{attribute 'GeneratedUsingTerminal: EL6070-0000-0016'}
{attribute addProperty BoxType "EL6070-0000-0016"}
{attribute addProperty Id "InfoDataAT %I*InfoData_32EB74EA10"}
{attribute addProperty CRC "4004708084"}
{attribute addProperty Size "10"}
TYPE EL6070_EEB2FEF4 EXTENDS EtcSlaveTerminalBase_947E5A46 :
STRUCT
	{attribute addProperty Name "InfoData"}
	InfoData : InfoData_32EB74EA;
END_STRUCT
END_TYPE

(* stored: Version 1.2.0.0, ProductVersion 3.1.4024.9
   DUT EL6070_EEB2FEF4: Id {4efff1e7-fe69-4162-825a-c733cd3a4e45} *)
